INTERFACE I_DigitalOut

METHOD M_On
VAR_INPUT
END_VAR
END_METHOD

 METHOD M_Off
VAR_INPUT
END_VAR
END_METHOD

END_INTERFACE

(* stored: Version 1.1.0.1, ProductVersion 3.1.0.19
   Itf I_DigitalOut: Id {8c5a6691-9636-489a-85c3-2c926edf1d80}
   Method M_On: Id {3a7646a9-3cb5-40c8-8e2b-04cade896a0b}
   Method M_Off: Id {899ffef1-0829-4a26-8138-7293424e86b0} *)
